(* IEC 61131-3 sources: CodesysTest/export/Function Blocks/SolenoidValves/FB_VacuumGenerator.pou, 3 files *)

(* ---- FB_VacuumGenerator.pou.st ---- *)
(*#-#-#-#-#-#-#-#-#-#---Declaration---#-#-#-#-#-#-#-#-#-#-#-#-#*)

FUNCTION_BLOCK FB_VacuumGenerator EXTENDS FB_SolenoidValve
VAR_INPUT
END_VAR
VAR_OUTPUT
END_VAR
VAR
END_VAR
(*#-#-#-#-#-#-#-#-#-#---Implementation---#-#-#-#-#-#-#-#-#-#-#-#-#*)

(* ---- GeneratorsOff.m.st ---- *)
(*#-#-#-#-#-#-#-#-#-#---Declaration---#-#-#-#-#-#-#-#-#-#-#-#-#*)

METHOD GeneratorsOff
VAR_INPUT
END_VAR
(*#-#-#-#-#-#-#-#-#-#---Implementation---#-#-#-#-#-#-#-#-#-#-#-#-#*)

THIS^.solenoid0 := FALSE;
THIS^.solenoid1 := FALSE;

(* ---- GeneratorsOn.m.st ---- *)
(*#-#-#-#-#-#-#-#-#-#---Declaration---#-#-#-#-#-#-#-#-#-#-#-#-#*)

METHOD GeneratorsOn
VAR_INPUT
END_VAR
(*#-#-#-#-#-#-#-#-#-#---Implementation---#-#-#-#-#-#-#-#-#-#-#-#-#*)

THIS^.solenoid0 := TRUE;
THIS^.solenoid1 := FALSE;
